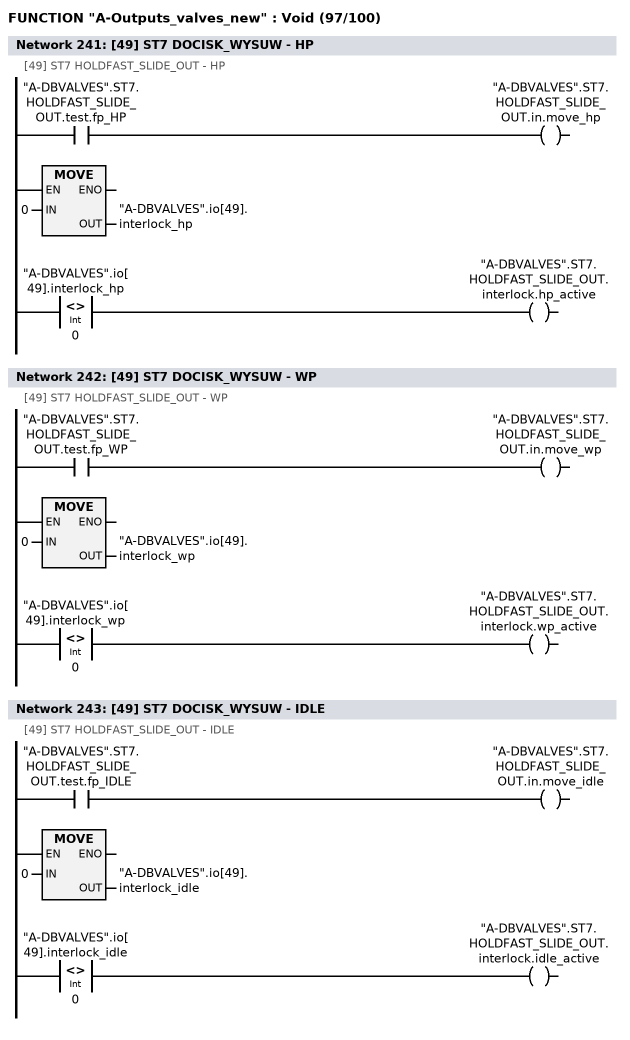
      O "A-DBVALVES".ST7.HOLDFAST_SLIDE_OUT.test.fp_HP;
//    O     "A-Flags".STATION.IN_HP_STEP
      = "A-DBVALVES".ST7.HOLDFAST_SLIDE_OUT.in.move_hp;

// Interlock hp
      L 0;
      T "A-DBVALVES".io[49].interlock_hp;

//{INTERLOCK_HP49}

      A(;
      L "A-DBVALVES".io[49].interlock_hp;
      L 0;
      <>I;
      );
      = "A-DBVALVES".ST7.HOLDFAST_SLIDE_OUT.interlock.hp_active;
NETWORK
TITLE = [49] ST7 DOCISK_WYSUW - WP
//[49] ST7 HOLDFAST_SLIDE_OUT - WP
      O "A-DBVALVES".ST7.HOLDFAST_SLIDE_OUT.test.fp_WP;
      = "A-DBVALVES".ST7.HOLDFAST_SLIDE_OUT.in.move_wp;

// Interlock wp
      L 0;
      T "A-DBVALVES".io[49].interlock_wp;

//{INTERLOCK_WP49}

      A(;
      L "A-DBVALVES".io[49].interlock_wp;
      L 0;
      <>I;
      );
      = "A-DBVALVES".ST7.HOLDFAST_SLIDE_OUT.interlock.wp_active;
NETWORK
TITLE = [49] ST7 DOCISK_WYSUW - IDLE
//[49] ST7 HOLDFAST_SLIDE_OUT - IDLE
      O "A-DBVALVES".ST7.HOLDFAST_SLIDE_OUT.test.fp_IDLE;
      = "A-DBVALVES".ST7.HOLDFAST_SLIDE_OUT.in.move_idle;

// Interlock idle
      L 0;
      T "A-DBVALVES".io[49].interlock_idle;

//{INTERLOCK_IDLE49}

      A(;
      L "A-DBVALVES".io[49].interlock_idle;
      L 0;
      <>I;
      );
      = "A-DBVALVES".ST7.HOLDFAST_SLIDE_OUT.interlock.idle_active;
NETWORK
TITLE = [49] ST7 DOCISK_WYSUW
//[49] ST7 HOLDFAST_SLIDE_OUT
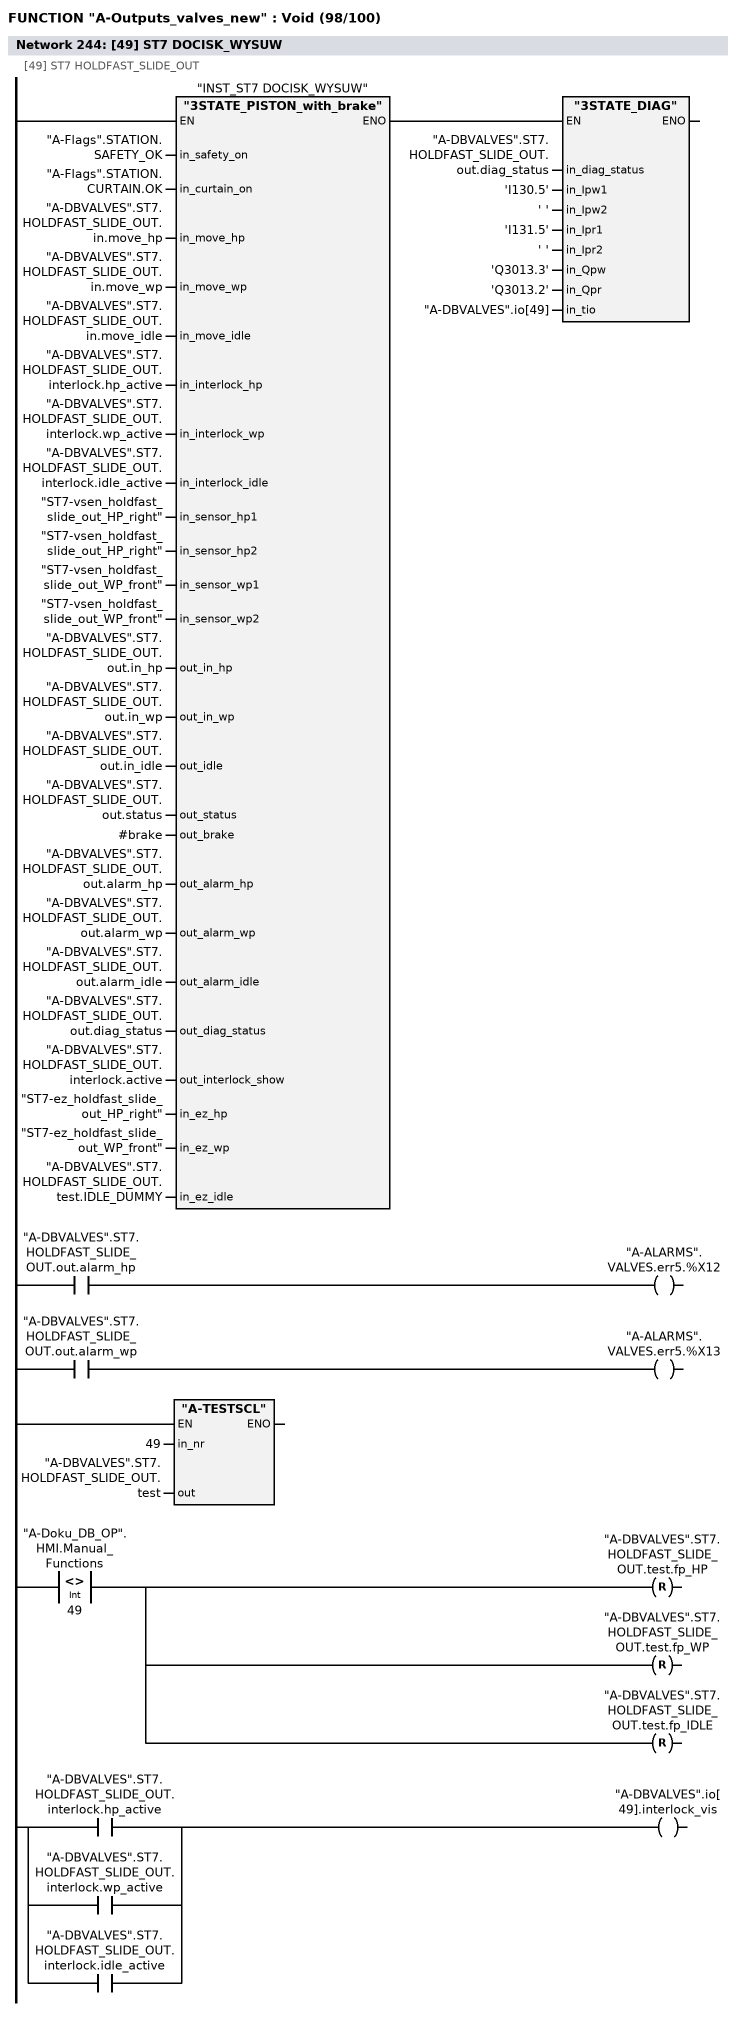
      CALL "3STATE_PISTON_with_brake", "INST_ST7 DOCISK_WYSUW"
      (  in_safety_on                := "A-Flags".STATION.SAFETY_OK ,
         in_curtain_on               := "A-Flags".STATION.CURTAIN.OK ,
         in_move_hp                  := "A-DBVALVES".ST7.HOLDFAST_SLIDE_OUT.in.move_hp ,
         in_move_wp                  := "A-DBVALVES".ST7.HOLDFAST_SLIDE_OUT.in.move_wp ,
         in_move_idle                := "A-DBVALVES".ST7.HOLDFAST_SLIDE_OUT.in.move_idle ,
         in_interlock_hp             := "A-DBVALVES".ST7.HOLDFAST_SLIDE_OUT.interlock.hp_active ,
         in_interlock_wp             := "A-DBVALVES".ST7.HOLDFAST_SLIDE_OUT.interlock.wp_active ,
         in_interlock_idle           := "A-DBVALVES".ST7.HOLDFAST_SLIDE_OUT.interlock.idle_active ,
         in_sensor_hp1               := "ST7-vsen_holdfast_slide_out_HP_right" ,
         in_sensor_hp2               := "ST7-vsen_holdfast_slide_out_HP_right" ,
         in_sensor_wp1               := "ST7-vsen_holdfast_slide_out_WP_front" ,
         in_sensor_wp2               := "ST7-vsen_holdfast_slide_out_WP_front" ,
         out_in_hp                   := "A-DBVALVES".ST7.HOLDFAST_SLIDE_OUT.out.in_hp ,
         out_in_wp                   := "A-DBVALVES".ST7.HOLDFAST_SLIDE_OUT.out.in_wp ,
         out_idle                    := "A-DBVALVES".ST7.HOLDFAST_SLIDE_OUT.out.in_idle ,
         out_status                  := "A-DBVALVES".ST7.HOLDFAST_SLIDE_OUT.out.status ,
         out_brake                   := #brake ,
         out_alarm_hp                := "A-DBVALVES".ST7.HOLDFAST_SLIDE_OUT.out.alarm_hp ,
         out_alarm_wp                := "A-DBVALVES".ST7.HOLDFAST_SLIDE_OUT.out.alarm_wp ,
         out_alarm_idle              := "A-DBVALVES".ST7.HOLDFAST_SLIDE_OUT.out.alarm_idle ,
         out_diag_status             := "A-DBVALVES".ST7.HOLDFAST_SLIDE_OUT.out.diag_status ,
         out_interlock_show          := "A-DBVALVES".ST7.HOLDFAST_SLIDE_OUT.interlock.active ,
         in_ez_hp                    := "ST7-ez_holdfast_slide_out_HP_right" ,
         in_ez_wp                    := "ST7-ez_holdfast_slide_out_WP_front" ,
         in_ez_idle                  := "A-DBVALVES".ST7.HOLDFAST_SLIDE_OUT.test.IDLE_DUMMY
      );

      CALL "3STATE_DIAG"
      (  in_diag_status              := "A-DBVALVES".ST7.HOLDFAST_SLIDE_OUT.out.diag_status ,
         in_Ipw1                     := 'I130.5' ,
         in_Ipw2                     := ' ' ,
         in_Ipr1                     := 'I131.5' ,
         in_Ipr2                     := ' ' ,
         in_Qpw                      := 'Q3013.3' ,
         in_Qpr                      := 'Q3013.2' ,
         in_tio                      := "A-DBVALVES".io[49]
      );

      A "A-DBVALVES".ST7.HOLDFAST_SLIDE_OUT.out.alarm_hp;
      = "A-ALARMS".VALVES.err5.%X12;

      A "A-DBVALVES".ST7.HOLDFAST_SLIDE_OUT.out.alarm_wp;
      = "A-ALARMS".VALVES.err5.%X13;

      CALL "A-TESTSCL"
      (  in_nr                       := 49 ,
         out                         := "A-DBVALVES".ST7.HOLDFAST_SLIDE_OUT.test
      );

      A(;
      L "A-Doku_DB_OP".HMI.Manual_Functions;
      L 49;
      <>I;
      );
      R "A-DBVALVES".ST7.HOLDFAST_SLIDE_OUT.test.fp_HP;
      R "A-DBVALVES".ST7.HOLDFAST_SLIDE_OUT.test.fp_WP;
      R "A-DBVALVES".ST7.HOLDFAST_SLIDE_OUT.test.fp_IDLE;

      O "A-DBVALVES".ST7.HOLDFAST_SLIDE_OUT.interlock.hp_active;
      O "A-DBVALVES".ST7.HOLDFAST_SLIDE_OUT.interlock.wp_active;
      O "A-DBVALVES".ST7.HOLDFAST_SLIDE_OUT.interlock.idle_active;
      = "A-DBVALVES".io[49].interlock_vis;
NETWORK
TITLE = -

NETWORK
TITLE = [50] ST7 DOCISK - HP
//[50] ST7 HOLDFAST - HP
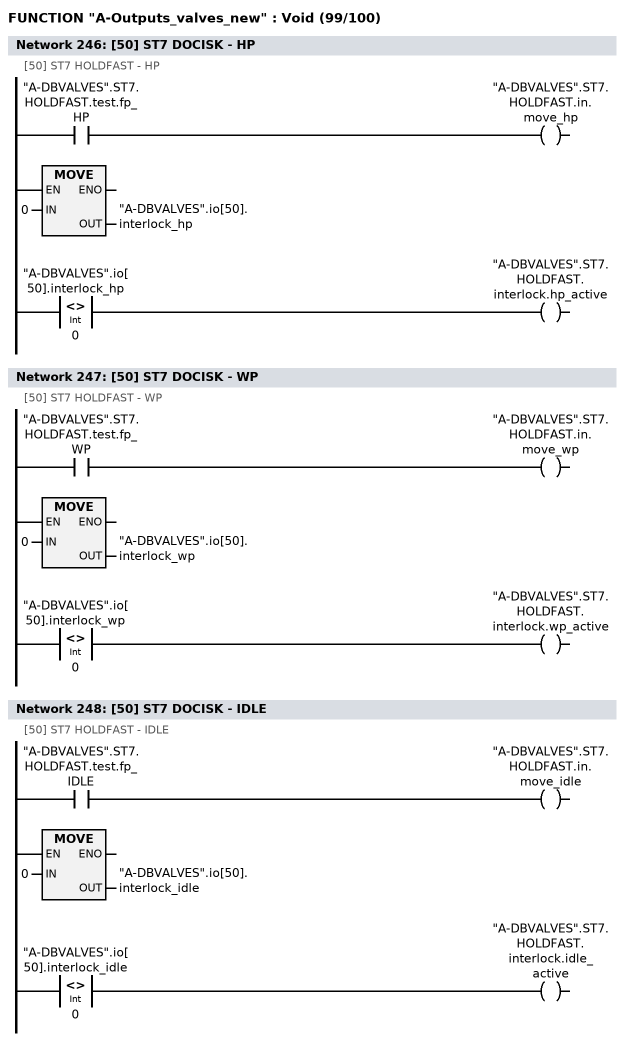
      O "A-DBVALVES".ST7.HOLDFAST.test.fp_HP;
//    O     "A-Flags".STATION.IN_HP_STEP
      = "A-DBVALVES".ST7.HOLDFAST.in.move_hp;

// Interlock hp
      L 0;
      T "A-DBVALVES".io[50].interlock_hp;

//{INTERLOCK_HP50}

      A(;
      L "A-DBVALVES".io[50].interlock_hp;
      L 0;
      <>I;
      );
      = "A-DBVALVES".ST7.HOLDFAST.interlock.hp_active;
NETWORK
TITLE = [50] ST7 DOCISK - WP
//[50] ST7 HOLDFAST - WP
      O "A-DBVALVES".ST7.HOLDFAST.test.fp_WP;
      = "A-DBVALVES".ST7.HOLDFAST.in.move_wp;

// Interlock wp
      L 0;
      T "A-DBVALVES".io[50].interlock_wp;

//{INTERLOCK_WP50}

      A(;
      L "A-DBVALVES".io[50].interlock_wp;
      L 0;
      <>I;
      );
      = "A-DBVALVES".ST7.HOLDFAST.interlock.wp_active;
NETWORK
TITLE = [50] ST7 DOCISK - IDLE
//[50] ST7 HOLDFAST - IDLE
      O "A-DBVALVES".ST7.HOLDFAST.test.fp_IDLE;
      = "A-DBVALVES".ST7.HOLDFAST.in.move_idle;

// Interlock idle
      L 0;
      T "A-DBVALVES".io[50].interlock_idle;

//{INTERLOCK_IDLE50}

      A(;
      L "A-DBVALVES".io[50].interlock_idle;
      L 0;
      <>I;
      );
      = "A-DBVALVES".ST7.HOLDFAST.interlock.idle_active;
NETWORK
TITLE = [50] ST7 DOCISK
//[50] ST7 HOLDFAST
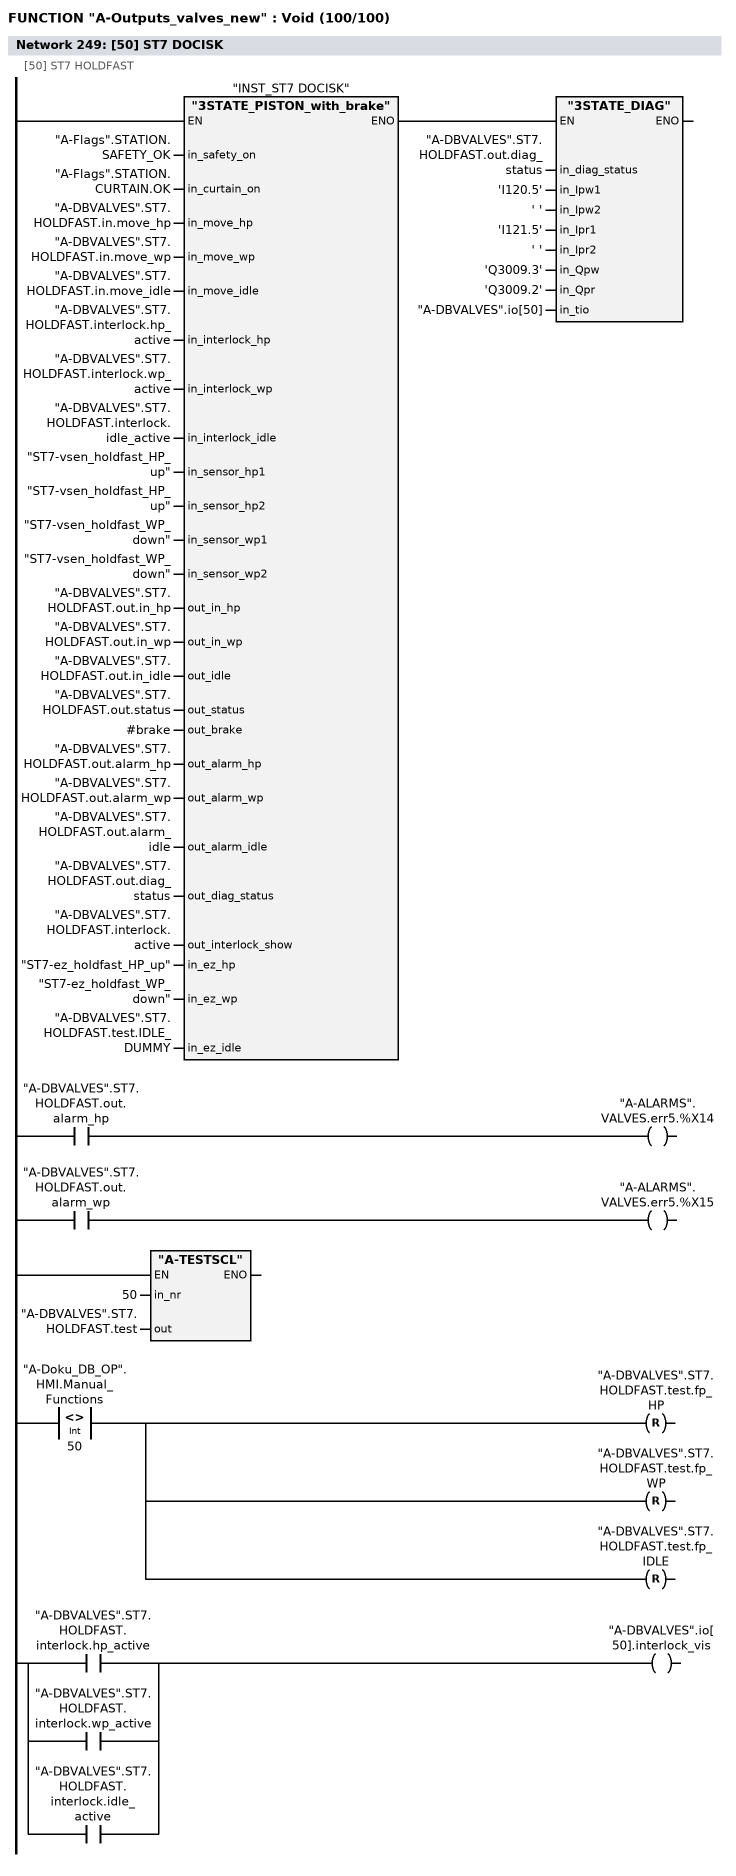
      CALL "3STATE_PISTON_with_brake", "INST_ST7 DOCISK"
      (  in_safety_on                := "A-Flags".STATION.SAFETY_OK ,
         in_curtain_on               := "A-Flags".STATION.CURTAIN.OK ,
         in_move_hp                  := "A-DBVALVES".ST7.HOLDFAST.in.move_hp ,
         in_move_wp                  := "A-DBVALVES".ST7.HOLDFAST.in.move_wp ,
         in_move_idle                := "A-DBVALVES".ST7.HOLDFAST.in.move_idle ,
         in_interlock_hp             := "A-DBVALVES".ST7.HOLDFAST.interlock.hp_active ,
         in_interlock_wp             := "A-DBVALVES".ST7.HOLDFAST.interlock.wp_active ,
         in_interlock_idle           := "A-DBVALVES".ST7.HOLDFAST.interlock.idle_active ,
         in_sensor_hp1               := "ST7-vsen_holdfast_HP_up" ,
         in_sensor_hp2               := "ST7-vsen_holdfast_HP_up" ,
         in_sensor_wp1               := "ST7-vsen_holdfast_WP_down" ,
         in_sensor_wp2               := "ST7-vsen_holdfast_WP_down" ,
         out_in_hp                   := "A-DBVALVES".ST7.HOLDFAST.out.in_hp ,
         out_in_wp                   := "A-DBVALVES".ST7.HOLDFAST.out.in_wp ,
         out_idle                    := "A-DBVALVES".ST7.HOLDFAST.out.in_idle ,
         out_status                  := "A-DBVALVES".ST7.HOLDFAST.out.status ,
         out_brake                   := #brake ,
         out_alarm_hp                := "A-DBVALVES".ST7.HOLDFAST.out.alarm_hp ,
         out_alarm_wp                := "A-DBVALVES".ST7.HOLDFAST.out.alarm_wp ,
         out_alarm_idle              := "A-DBVALVES".ST7.HOLDFAST.out.alarm_idle ,
         out_diag_status             := "A-DBVALVES".ST7.HOLDFAST.out.diag_status ,
         out_interlock_show          := "A-DBVALVES".ST7.HOLDFAST.interlock.active ,
         in_ez_hp                    := "ST7-ez_holdfast_HP_up" ,
         in_ez_wp                    := "ST7-ez_holdfast_WP_down" ,
         in_ez_idle                  := "A-DBVALVES".ST7.HOLDFAST.test.IDLE_DUMMY
      );

      CALL "3STATE_DIAG"
      (  in_diag_status              := "A-DBVALVES".ST7.HOLDFAST.out.diag_status ,
         in_Ipw1                     := 'I120.5' ,
         in_Ipw2                     := ' ' ,
         in_Ipr1                     := 'I121.5' ,
         in_Ipr2                     := ' ' ,
         in_Qpw                      := 'Q3009.3' ,
         in_Qpr                      := 'Q3009.2' ,
         in_tio                      := "A-DBVALVES".io[50]
      );

      A "A-DBVALVES".ST7.HOLDFAST.out.alarm_hp;
      = "A-ALARMS".VALVES.err5.%X14;

      A "A-DBVALVES".ST7.HOLDFAST.out.alarm_wp;
      = "A-ALARMS".VALVES.err5.%X15;

      CALL "A-TESTSCL"
      (  in_nr                       := 50 ,
         out                         := "A-DBVALVES".ST7.HOLDFAST.test
      );

      A(;
      L "A-Doku_DB_OP".HMI.Manual_Functions;
      L 50;
      <>I;
      );
      R "A-DBVALVES".ST7.HOLDFAST.test.fp_HP;
      R "A-DBVALVES".ST7.HOLDFAST.test.fp_WP;
      R "A-DBVALVES".ST7.HOLDFAST.test.fp_IDLE;

      O "A-DBVALVES".ST7.HOLDFAST.interlock.hp_active;
      O "A-DBVALVES".ST7.HOLDFAST.interlock.wp_active;
      O "A-DBVALVES".ST7.HOLDFAST.interlock.idle_active;
      = "A-DBVALVES".io[50].interlock_vis;
NETWORK
TITLE = -


END_FUNCTION

